KUKA KRL data list: dockof_2.dat

&ACCESS RV1
&REL 140
&COMMENT PLACE GUN 2
DEFDAT  DOCKOF_2
;FOLD EXTERNAL DECLARATIONS;%{PE}%MKUKATPBASIS,%CEXT,%VCOMMON,%P
;FOLD GRIPPERTECH EXT
EXT  H50 (INT  :IN,INT  :IN,INT  :IN,GRP_TYP  :IN )
;ENDFOLD (GRIPPERTECH EXT)
;FOLD SPOTTECH EXT
EXT  USERSPOT (S_COMMAND  :IN,SPOT_TYPE  :IN )
;ENDFOLD (SPOTTECH EXT)
;FOLD BASISTECH EXT;%{PE}%MKUKATPBASIS,%CEXT,%VEXT,%P
EXT  BAS (BAS_COMMAND  :IN,REAL  :IN )
DECL INT SUCCESS
;ENDFOLD (BASISTECH EXT)
;FOLD USER EXT;%{E}%MKUKATPUSER,%CEXT,%VEXT,%P
;Make here your modifications
;ENDFOLD (USER EXT)
;ENDFOLD (EXTERNAL DECLERATIONS)
;*      FDAT Declarations     *

;******************************
;*     E6POS Declarations     *
;******************************

DECL E6POS XP10={X -981.764771,Y 1883.28101,Z 561.632813,A -85.3195038,B 0.149295896,C -0.627375901,S 2,T 43,E1 -735.495178,E2 0.0,E3 0.0,E4 0.0,E5 0.0,E6 0.0}
DECL E6POS XP20={X -1295.61206,Y 1934.646,Z 42.0023003,A -85.3188019,B 0.147270799,C -0.629731119,S 2,T 43,E1 -735.49353,E2 0.0,E3 0.0,E4 0.0,E5 0.0,E6 0.0}
DECL E6POS XP30={X -1415.08899,Y 1875.94202,Z -601.858826,A -85.3188095,B 0.148737103,C -0.630693614,S 2,T 43,E1 -735.491699,E2 0.0,E3 0.0,E4 0.0,E5 0.0,E6 0.0}
DECL E6POS XP40={X -1439.323,Y 1875.89795,Z -630.582214,A -84.2455215,B 0.0450858884,C -0.629668415,S 2,T 43,E1 -735.49353,E2 0.0,E3 0.0,E4 0.0,E5 0.0,E6 0.0}
DECL E6POS XP50={X -1439.32996,Y 1875.90295,Z -670.736511,A -84.2452698,B 0.0452245101,C -0.629822373,S 2,T 43,E1 -735.49353,E2 0.0,E3 0.0,E4 0.0,E5 0.0,E6 0.0}
DECL E6POS XP60={X -1414.71301,Y 1875.07996,Z 706.503113,A -134.240997,B -0.652029216,C 179.492798,S 2,T 43,E1 -735.497009,E2 0.0,E3 0.0,E4 0.0,E5 0.0,E6 0.0}
DECL E6POS XP70={X -1416.05505,Y 1879.71399,Z 712.868896,A -135.317596,B -0.386982203,C 179.484802,S 2,T 43,E1 -735.491699,E2 0.0,E3 0.0,E4 0.0,E5 0.0,E6 0.0}
DECL E6POS XP80={X -1127.36902,Y 2445.76807,Z 816.869385,A -45.7330017,B 0.4947837,C 179.7724,S 2,T 11,E1 -1181.96399,E2 0.0,E3 0.0,E4 0.0,E5 0.0,E6 0.0}

;******************************
;*     FDAT Declarations      *
;******************************

DECL FDAT FP10={TOOL_NO 2,BASE_NO 0,IPO_FRAME #BASE}
DECL FDAT FP20={TOOL_NO 2,BASE_NO 0,IPO_FRAME #BASE}
DECL FDAT FP30={TOOL_NO 2,BASE_NO 0,IPO_FRAME #BASE}
DECL FDAT FP40={TOOL_NO 2,BASE_NO 0,IPO_FRAME #BASE}
DECL FDAT FP50={TOOL_NO 2,BASE_NO 0,IPO_FRAME #BASE}
DECL FDAT FP60={TOOL_NO 14,BASE_NO 0,IPO_FRAME #BASE}
DECL FDAT FP70={TOOL_NO 10,BASE_NO 0,IPO_FRAME #BASE}
DECL FDAT FP80={TOOL_NO 10,BASE_NO 0,IPO_FRAME #BASE}

;******************************
;*  PDAT & LDAT Declarations  *
;******************************

DECL PDAT PH={VEL 100.0,ACC 100.0,APO_DIST 100.0}
DECL LDAT LH={VEL 2.0,ACC 100.0,APO_DIST 100.0,APO_FAC 50.0,ORI_TYP #VAR}

DECL PDAT PPDAT1={VEL 100.0,ACC 100.0,APO_DIST 100.0}
DECL E6POS XP1={X -1394.16199,Y 1902.81897,Z -524.886108,A -85.3188629,B 0.148389801,C -0.63038218,S 2,T 43,E1 -735.491699,E2 0.0,E3 0.0,E4 0.0,E5 0.0,E6 0.0}
DECL FDAT FP1={TOOL_NO 2,BASE_NO 0,IPO_FRAME #BASE,POINT2[] " "}
ENDDAT
